//---------------------------------------------------------------------------------------------------------------
//
//  HAUD 2025.02.24
//
//  - EXAMPLE, change, adapt, use
//  -----------------------------
//  - processes and top level workflow examples
//  - based on fb_Instance for processes
//  - fb_Application as top level control for starting, stopping, restarting etc..
//---------------------------------------------------------------------------------------------------------------
PROGRAM MAIN_APP
VAR
  eInit                       : E_PROGRESS;   // application startup state info
  nProcess                    : uint;

  tonWriteLog                 : Tc2_Standard.TON;
  tWriteLog                   : TIME := T#1S;

  stMsg                       : ST_Message;

  _nBufferOutfeedTarget       : ARRAY[1..2] OF E_INSTANCE;
  _nStnFrst                   : UDINT;

  eMsgState                   : e_message_state;
  eMsgProgress                : E_PROGRESS;
END_VAR

//-----------------------------------------------------------------------------------------------------------------
//-----------------------------------------------------------------------------------------------------------------
// check for MAIN.eInit
//  - wait for fb_TransportUnit to be fully started up
//-----------------------------------------------------------------------------------------------------------------
IF NOT (MAIN.eInit = E_PROGRESS.PROGRESS_DONE) 
THEN 
  eInit                                                     := E_PROGRESS.PROGRESS_INVALID; 
  FOR nProcess := E_INSTANCE.BUFFER_INFEED TO MAX_PROCESS
  DO
    GVL_MSG.MessageLevelProcess[nProcess]                   := GVL_MSG.MessageLevel;
  END_FOR
  //ApplicationMain.MessageLevel                              := GVL_MSG.MessageLevel;

  RETURN; 
END_IF
//-----------------------------------------------------------------------------------------------------------------
// set MAIN_APP message device identification
//-----------------------------------------------------------------------------------------------------------------
stMsg.eDevice                                               := e_Device.Application;
//-----------------------------------------------------------------------------------------------------------------
//-----------------------------------------------------------------------------------------------------------------
//-----------------------------------------------------------------------------------------------------------------
// /assign dataflow
//-----------------------------------------------------------------------------------------------------------------
FOR nProcess := 1 TO MAX_PROCESS
DO
  // identification for inter-process-commands and process ST_MESSAGE.eDevice
  GVL_APPLICATION.ProcessCollector[nProcess].ProcessId      :=    nProcess;

  // linked list for you to use for inter-process-commands (start trigger, exit trigger..)
  GVL_APPLICATION.ItfProcessList[nProcess]                  :=    GVL_APPLICATION.ProcessList[nProcess];

  // give reference of all XtsStations to every process; range of process must be set at startup (see action Init())
  GVL_APPLICATION.ProcessCollector[nProcess].StationCtrl    REF=  GVL_XTS.StationCtrl;
  GVL_APPLICATION.ProcessCollector[nProcess].StationState   REF=  GVL_XTS.StationState;

  GVL_APPLICATION.ProcessCollector[nProcess].MoverInfo      REF=  GVL_XTS.MoverInfo;

  // global interfaces for you to use in your process function blocks
  GVL_APPLICATION.ItfProcessCollector[nProcess]             :=    GVL_APPLICATION.ProcessCollector[nProcess];
END_FOR
//-----------------------------------------------------------------------------------------------------------------
//-----------------------------------------------------------------------------------------------------------------
//-----------------------------------------------------------------------------------------------------------------
//  process instances
//-----------------------------------------------------------------------------------------------------------------
GVL_APPLICATION.TicketControl.ItfList                          :=    GVL_APPLICATION.TicketList;
GVL_APPLICATION.TicketControl.Ctrl                             REF=  GVL_APPLICATION.TicketListControl;
GVL_APPLICATION.TicketControl.State                            REF=  GVL_APPLICATION.TicketListState;
GVL_APPLICATION.TicketControl.NodeDataInput                    REF=  GVL_APPLICATION.TicketListDataInput;
GVL_APPLICATION.TicketControl.NodeDataOutput                   REF=  GVL_APPLICATION.TicketListDataOutput;
GVL_APPLICATION.TicketControl.MessageLevel                     :=    GVL_MSG.MessageLevelProcess[e_instance.PROCESS_CONDUCTOR];

GVL_APPLICATION.ProcessConductor.TicketLinkedList           :=    GVL_APPLICATION.TicketList;
GVL_APPLICATION.ProcessConductor.InstanceCtrl               REF=  GVL_APPLICATION.InstanceCtrl;
GVL_APPLICATION.ProcessConductor.InstanceState              REF=  GVL_APPLICATION.InstanceState;
GVL_APPLICATION.ProcessConductor.MessageLevel               :=    GVL_MSG.MessageLevelProcess[e_instance.PROCESS_CONDUCTOR];

GVL_APPLICATION.BufferInfeed.InstanceCtrl                   REF=  GVL_APPLICATION.InstanceCtrl;
GVL_APPLICATION.BufferInfeed.InstanceState                  REF=  GVL_APPLICATION.InstanceState;
GVL_APPLICATION.BufferInfeed.MessageLevel                   :=    GVL_MSG.MessageLevelProcess[e_instance.BUFFER_INFEED];
                                                            
GVL_APPLICATION.Infeed.InstanceCtrl                         REF=  GVL_APPLICATION.InstanceCtrl;
GVL_APPLICATION.Infeed.InstanceState                        REF=  GVL_APPLICATION.InstanceState;
GVL_APPLICATION.Infeed.MessageLevel                         :=    E_MessageType.eMessageSentient; //GVL_MSG.MessageLevelProcess[e_instance.INFEED];
                                                            
GVL_APPLICATION.BufferOutfeed.InstanceCtrl                  REF=  GVL_APPLICATION.InstanceCtrl;
GVL_APPLICATION.BufferOutfeed.InstanceState                 REF=  GVL_APPLICATION.InstanceState;
GVL_APPLICATION.BufferOutfeed.MessageLevel                  :=    GVL_MSG.MessageLevelProcess[e_instance.BUFFER_OUTFEED];
                                                            
GVL_APPLICATION.Outfeed_R1.InstanceCtrl                     REF=  GVL_APPLICATION.InstanceCtrl;
GVL_APPLICATION.Outfeed_R1.InstanceState                    REF=  GVL_APPLICATION.InstanceState;
GVL_APPLICATION.Outfeed_R1.MessageLevel                     :=    GVL_MSG.MessageLevelProcess[e_instance.OUTFEED_ROBOT_R1];
                                                            
GVL_APPLICATION.Outfeed_R2.InstanceCtrl                     REF=  GVL_APPLICATION.InstanceCtrl;
GVL_APPLICATION.Outfeed_R2.InstanceState                    REF=  GVL_APPLICATION.InstanceState;
GVL_APPLICATION.Outfeed_R2.MessageLevel                     :=    GVL_MSG.MessageLevelProcess[e_instance.OUTFEED_ROBOT_R2];
                                                            
GVL_APPLICATION.SenderFast.InstanceCtrl                     REF=  GVL_APPLICATION.InstanceCtrl;
GVL_APPLICATION.SenderFast.InstanceState                    REF=  GVL_APPLICATION.InstanceState;
GVL_APPLICATION.SenderFast.MessageLevel                     :=    GVL_MSG.MessageLevelProcess[e_instance.SENDER_FAST];
                                                            
GVL_APPLICATION.SenderBufferInfeed.InstanceCtrl             REF=  GVL_APPLICATION.InstanceCtrl;
GVL_APPLICATION.SenderBufferInfeed.InstanceState            REF=  GVL_APPLICATION.InstanceState;
GVL_APPLICATION.SenderBufferInfeed.MessageLevel             :=    GVL_MSG.MessageLevelProcess[e_instance.SENDER_BUFFER_INFEED];
//-----------------------------------------------------------------------------------------------------------------
//-----------------------------------------------------------------------------------------------------------------
//-----------------------------------------------------------------------------------------------------------------
//  main application class
//-----------------------------------------------------------------------------------------------------------------
(*
GVL_APPLICATION.ApplicationMain.Ctrl                        REF=  GVL_APPLICATION.AppControl;
GVL_APPLICATION.ApplicationMain.State                       REF=  GVL_APPLICATION.AppState;
GVL_APPLICATION.ApplicationMain.CollectorInterface          REF=  GVL_APPLICATION.ItfProcessCollector;
GVL_APPLICATION.ApplicationMain.ProcessLinkedLists          REF=  GVL_APPLICATION.ItfProcessList;
GVL_APPLICATION.ApplicationMain.XtsTransportCtrl            REF=  GVL_XTS.XtsTransportCtrl;
GVL_APPLICATION.ApplicationMain.XtsTransportState           REF=  GVL_XTS.XtsTransportState;
GVL_APPLICATION.ApplicationMain.InstanceCtrl                REF=  GVL_APPLICATION.InstanceCtrl;
GVL_APPLICATION.ApplicationMain.InstanceState               REF=  GVL_APPLICATION.InstanceState;
*)
//-----------------------------------------------------------------------------------------------------------------
//-----------------------------------------------------------------------------------------------------------------
//-----------------------------------------------------------------------------------------------------------------
// assign dataflow/
//-----------------------------------------------------------------------------------------------------------------
//-----------------------------------------------------------------------------------------------------------------
//-----------------------------------------------------------------------------------------------------------------
//-----------------------------------------------------------------------------------------------------------------
//  /STARTUP
//
// startup procedure for application
//  - connects processes and XtsStations
//-----------------------------------------------------------------------------------------------------------------
CASE eInit
OF
  E_PROGRESS.PROGRESS_INVALID:                // first cycle startup
    //---------------------------------------------------------------------------------------------------------------
    // first cycle startup
    // - wait for extern to give the command, if we are waiting here MAIN is ready, extern can see that
    //---------------------------------------------------------------------------------------------------------------
    GVL_MSG.ApplicationMessageCtrl.Cmd        := E_MESSAGE_CTRL.MSG_CTRL_NULL;
    eInit                                     := E_PROGRESS.PROGRESS_INIT;

  E_PROGRESS.PROGRESS_INIT:
    //---------------------------------------------------------------------------------------------------------------
    // wait for extern to select valid variant
    //---------------------------------------------------------------------------------------------------------------
    CASE GVL_APPLICATION.AppControl.Variant
    OF
      E_APP_VARIANT.VARIANT_OUTPUT_24:
        eInit                                 := E_PROGRESS.PROGRESS_BUSY;
        ProcessInit_R1R2();
  
        stMsg.eType                           := E_MessageType.eMessageInfo;
        stMsg.eSubdevice                      := e_Subdevice.General;
        stMsg.iErrorNumber                    := eInit;
        stMsg.sText                           := concat('MAIN_APP.eInit: ', TO_STRING(eInit));
        stMsg.sText                           := concat(stMsg.sText, ': ');
        stMsg.sText                           := concat(stMsg.sText, TO_STRING(E_INSTANCE.OUTFEED_ROBOT_R1));
        stMsg.sText                           := concat(stMsg.sText, ': ');
        stMsg.sText                           := concat(stMsg.sText, TO_STRING(E_INSTANCE.OUTFEED_ROBOT_R2));
        f_MessageSet(stMsg);

      E_APP_VARIANT.VARIANT_OUTPUT_CLAMP:
        eInit                                 := E_PROGRESS.PROGRESS_BUSY;
        ProcessInit_CLAMP();
  
        stMsg.eType                           := E_MessageType.eMessageInfo;
        stMsg.eSubdevice                      := e_Subdevice.General;
        stMsg.iErrorNumber                    := eInit;
        stMsg.sText                           := concat('MAIN_APP.eInit: ', TO_STRING(eInit));
        stMsg.sText                           := concat(stMsg.sText, ': ');
        stMsg.sText                           := concat(stMsg.sText, TO_STRING(E_INSTANCE.OUTFEED_ROBOT_R1));
        f_MessageSet(stMsg);
    END_CASE

  E_PROGRESS.PROGRESS_BUSY:
    //---------------------------------------------------------------------------------------------------------------
    // first cycle startup of all instances
    //---------------------------------------------------------------------------------------------------------------
    GVL_MSG.ApplicationMessageCtrl.Cmd        := E_MESSAGE_CTRL.MSG_CTRL_INIT;

    IF (GVL_MSG.ApplicationMessageState.State = E_MESSAGE_STATE.MSG_STATE_INIT + E_PROGRESS.PROGRESS_DONE)
    THEN
      eInit                                   := E_PROGRESS.PROGRESS_STARTUP;
    END_IF

  E_PROGRESS.PROGRESS_STARTUP:
    IF GVL_MSG.ApplicationMessageData.FileCreated
    THEN
      eInit                                   := E_PROGRESS.PROGRESS_DONE;
      GVL_MSG.ApplicationMessageCtrl.Cmd      := E_MESSAGE_CTRL.MSG_CTRL_NULL;
    END_IF
END_CASE
GVL_APPLICATION.AppState.AppInit              := eInit;
//-----------------------------------------------------------------------------------------------------------------
//-----------------------------------------------------------------------------------------------------------------
// STARTUP/
//-----------------------------------------------------------------------------------------------------------------
//-----------------------------------------------------------------------------------------------------------------
//-----------------------------------------------------------------------------------------------------------------
// /cyclic calls
//-----------------------------------------------------------------------------------------------------------------
//GVL_APPLICATION.ApplicationMain();

GVL_APPLICATION.TicketControl();

GVL_APPLICATION.ProcessConductor();
GVL_APPLICATION.BufferInfeed();
GVL_APPLICATION.Infeed();
GVL_APPLICATION.BufferOutfeed();
GVL_APPLICATION.Outfeed_R1();
GVL_APPLICATION.Outfeed_R2();
GVL_APPLICATION.SenderFast();
GVL_APPLICATION.SenderBufferInfeed();

FOR nProcess := 1 TO MAX_PROCESS
DO
  // cyclic interface check with XtsStations
  GVL_APPLICATION.ItfProcessCollector[nProcess].Cycle();    // collect XtsStation states, 
                                                            // manage ctrl input from process to XtsStations
END_FOR
//-----------------------------------------------------------------------------------------------------------------
//############################################################################
// /logging
//############################################################################
GVL_MSG.ApplicationMessageData.Ctrl           REF= GVL_MSG.ApplicationMessageCtrl;
GVL_MSG.ApplicationMessageData.State          REF= GVL_MSG.ApplicationMessageState;

GVL_MSG.ApplicationMessageData.MessageIndex   REF= GVL_MSG.MessageApplicationIndex;
GVL_MSG.ApplicationMessageData.ErrorIndex     REF= GVL_MSG.MessageApplicationError;

GVL_MSG.ApplicationMessageData.DirRoot        :=   ADR(GVL_MSG.LOG_DIR);
GVL_MSG.ApplicationMessageData.FileRoot       :=   ADR(GVL_MSG.LOG_FILE_APP);

GVL_MSG.ApplicationMessageData.MsgList        :=   ADR(GVL_MSG.ApplicationMessages);
GVL_MSG.ApplicationMessageData.LocalTime      :=   ADR(GVL_MSG.dtLocalTime);

GVL_MSG.ApplicationMessageData();

eMsgState                                     := f_GetState   (GVL_MSG.ApplicationMessageState.State);
eMsgProgress                                  := f_GetProgress(GVL_MSG.ApplicationMessageState.State);


CASE eMsgState
OF
  E_MESSAGE_STATE.MSG_STATE_NULL:
    CASE eMsgProgress
    OF
      E_PROGRESS.PROGRESS_INVALID:
        IF (GVL_MSG.MessageApplicationIndex > GVL_MSG.MAX_MESSAGE/100) OR
           (GVL_MSG.MessageApplicationError > 0)
        THEN
          GVL_MSG.ApplicationMessageCtrl.Cmd  := E_MESSAGE_CTRL.MSG_CTRL_WRITE;
        END_IF
    END_CASE

  E_MESSAGE_STATE.MSG_STATE_WRITE:
    CASE eMsgProgress
    OF
      E_PROGRESS.PROGRESS_ERROR,
      E_PROGRESS.PROGRESS_DONE:
        GVL_MSG.ApplicationMessageCtrl.Cmd    := E_MESSAGE_CTRL.MSG_CTRL_NULL;
    END_CASE

ELSE
    CASE eMsgProgress
    OF
      E_PROGRESS.PROGRESS_DONE:
        GVL_MSG.ApplicationMessageCtrl.Cmd    := E_MESSAGE_CTRL.MSG_CTRL_NULL;
    END_CASE
END_CASE
//############################################################################
// logging/
//############################################################################

ACTION ProcessInit_CLAMP:
//*************************************************************************************************************
//
// build configuration for Instances and ProcessInterfaces
//
//*************************************************************************************************************
//*************************************************************************************************************
// - ProcessConductor : Instance with connection to a cyclic linked list 
//                      Here does The Ticket with target processId and bitmask arrive 
//                      this instance forwards the ticket to its destination
//                        destination is BufferInfeed
//-------------------------------------------------------------------------------------------------------------
// whoami
//
// ticket box - transfersystem drops ticket
//-------------------------------------------------------------------------------------------------------------
ProcessConductor.ProcessId                := ProcessCollector[E_INSTANCE.PROCESS_CONDUCTOR].ProcessId;
ProcessConductor.CollectorInterface       := ItfProcessCollector;
ProcessConductor.ProcessLinkedLists       := ItfProcessList;

//*************************************************************************************************************
// - BufferInfeed     : single XtsStation which looks for input trigger from transfersystem, 
//                      transfersystem writes positions of XtsStations to be used at Infeed. 
//                      BufferInfeed is writing ItfProcessCollector[BufferInfeed.ProcessTarget].ActivateStation 
//                        for BufferInfeed target (Infeed / 12 XtsStations).
//                      BufferInfeed sends required amount of movers to WaitPos of XtsStations 
//                        of BufferInfeed target (Infeed / 12 XtsStations).
//-------------------------------------------------------------------------------------------------------------
// whoami
//
// process target (Infeed / 12 XtsStations)
//-------------------------------------------------------------------------------------------------------------
BufferInfeed.ProcessId                    := ProcessCollector[E_INSTANCE.BUFFER_INFEED].ProcessId;
BufferInfeed.ProcessTarget                := ProcessCollector[E_INSTANCE.INFEED].ProcessId;
BufferInfeed.CollectorInterface           := ItfProcessCollector;
BufferInfeed.ProcessLinkedLists           := ItfProcessList;
//-------------------------------------------------------------------------------------------------------------
// configure range of XtsStations for process
//
// see MAIN.StationParameterInit() for positions and dyn constraints
//-------------------------------------------------------------------------------------------------------------
ItfProcessCollector[BufferInfeed.ProcessId].StationFirst  := 53;
ItfProcessCollector[BufferInfeed.ProcessId].StationLast   := 53;

_nStnFrst                                 := ProcessCollector[BufferInfeed.ProcessId].StationFirst;
BufferInfeed.CheckPosition                := 15.0;

//-------------------------------------------------------------------------------------------------------------
//-------------------------------------------------------------------------------------------------------------
//*************************************************************************************************************
//*************************************************************************************************************
// - Infeed         : 12 XtsStations for transfersystem to unload
//                    Infeed is pulling in the movers according to list entry from BufferInfeed
//                    one stop only
//                    must be checked for all mover standstill in PosStop[1] of each XtsStation
//                    must be released by handshake from transfersystem (this is done by a TON for now)
//-------------------------------------------------------------------------------------------------------------
// whoami
//
// process target (BufferOutfeed / 1 XtsStation)
// TODO: 
//    configure infeed target for OUTFEED_CLAMP (12 XtsStations)
//    Infeed.ProcessTarget  := ProcessCollector[E_INSTANCE.OUTFEED_CLAMP].ProcessId;
//-------------------------------------------------------------------------------------------------------------
Infeed.ProcessId                          := ProcessCollector[E_INSTANCE.INFEED].ProcessId;
Infeed.ProcessTarget                      := ProcessCollector[E_INSTANCE.BUFFER_OUTFEED].ProcessId;
Infeed.CollectorInterface                 := ItfProcessCollector;
Infeed.ProcessLinkedLists                 := ItfProcessList;
//-------------------------------------------------------------------------------------------------------------
// configure range of XtsStations for process
//
// see MAIN.StationParameterInit() for positions and dyn constraints
//-------------------------------------------------------------------------------------------------------------
ItfProcessCollector[Infeed.ProcessId].StationFirst        :=  1;
ItfProcessCollector[Infeed.ProcessId].StationLast         := 12;
//-------------------------------------------------------------------------------------------------------------
//-------------------------------------------------------------------------------------------------------------
//*************************************************************************************************************
//*************************************************************************************************************
// - BufferOutfeed  : single XtsStation which distributes movers to specified range 
//                    Infeed sends all movers here 
//                    BufferOutfeed ensures that OutputR2 and OutputR1 have 12 movers each for every job
//                    BufferOutfeed checks if the Queue of this single XtsStation is empty or not
//-------------------------------------------------------------------------------------------------------------
// whoami
//
// process target (Outfeed (OutfeedR2 & OutfeedR1) / 24 XtsStations)
//
//  - optional process target (Outfeed 12 XtsStations)
//-------------------------------------------------------------------------------------------------------------
_nBufferOutfeedTarget[1] := E_INSTANCE.OUTFEED_ROBOT_R1;
_nBufferOutfeedTarget[2] := E_INSTANCE.OUTFEED_ROBOT_R1;

BufferOutfeed.ProcessId              := E_INSTANCE.BUFFER_OUTFEED;
BufferOutfeed.ProcessTarget          := _nBufferOutfeedTarget; 
BufferOutfeed.CollectorInterface     := ItfProcessCollector;
BufferOutfeed.ProcessLinkedLists     := ItfProcessList;
//-------------------------------------------------------------------------------------------------------------
// configure range of XtsStations for process
//
// see MAIN.StationParameterInit() for positions and dyn constraints
//-------------------------------------------------------------------------------------------------------------
ItfProcessCollector[BufferOutfeed.ProcessId].StationFirst  := 25;
ItfProcessCollector[BufferOutfeed.ProcessId].StationLast   := 25;

_nStnFrst                                 := ProcessCollector[BufferOutfeed.ProcessId].StationFirst;
BufferOutfeed.CheckPosition          := 2250.0;
//-------------------------------------------------------------------------------------------------------------
//-------------------------------------------------------------------------------------------------------------
//*************************************************************************************************************
//*************************************************************************************************************
// - Outfeed_R1  : 12 XtsStations for Robot 
//                    All XtsStations must be filled before robot can start 
//                    affter process all movers are sent to Sender process (high speed for the way back)
//                     
//                    
//-------------------------------------------------------------------------------------------------------------
// whoami
//
// process target (SenderFast / 1 XtsStation)
//-------------------------------------------------------------------------------------------------------------
Outfeed_R1.ProcessId                      := E_INSTANCE.OUTFEED_ROBOT_R1;
Outfeed_R1.ProcessTarget                  := ProcessCollector[E_INSTANCE.SENDER_FAST].ProcessId;
Outfeed_R1.CollectorInterface             := ItfProcessCollector;
Outfeed_R1.ProcessLinkedLists             := ItfProcessList;
//-------------------------------------------------------------------------------------------------------------
// configure range of XtsStations for process
//
// see MAIN.StationParameterInit() for positions and dyn constraints
//-------------------------------------------------------------------------------------------------------------
ItfProcessCollector[Outfeed_R1.ProcessId].StationFirst  := 13;
ItfProcessCollector[Outfeed_R1.ProcessId].StationLast   := 24;

_nStnFrst                                 := ProcessCollector[Outfeed_R1.ProcessId].StationFirst;
Outfeed_R1.CheckPosition                  := 2750.0;
//-------------------------------------------------------------------------------------------------------------
//-------------------------------------------------------------------------------------------------------------
//*************************************************************************************************************
//*************************************************************************************************************
// - Outfeed_R2  : 12 XtsStations for Robot 
//                    All XtsStations must be filled before robot can start 
//                    affter process all movers are sent to Sender process (high speed for the way back)
//                     
//                    
//-------------------------------------------------------------------------------------------------------------
// whoami
//
// process target (SenderFast / 1 XtsStation)
//-------------------------------------------------------------------------------------------------------------
Outfeed_R2.ProcessId                      := E_INSTANCE.OUTFEED_ROBOT_R2;
Outfeed_R2.ProcessTarget                  := ProcessCollector[E_INSTANCE.SENDER_FAST].ProcessId;
Outfeed_R2.CollectorInterface             := ItfProcessCollector;
Outfeed_R2.ProcessLinkedLists             := ItfProcessList;
//-------------------------------------------------------------------------------------------------------------
// configure range of XtsStations for process
//
// see MAIN.StationParameterInit() for positions and dyn constraints
//-------------------------------------------------------------------------------------------------------------
ItfProcessCollector[Outfeed_R2.ProcessId].StationFirst  := 38;
ItfProcessCollector[Outfeed_R2.ProcessId].StationLast   := 49;

_nStnFrst                                 := ProcessCollector[Outfeed_R2.ProcessId].StationFirst;
Outfeed_R2.CheckPosition                  := 6000.0;
//-------------------------------------------------------------------------------------------------------------
//-------------------------------------------------------------------------------------------------------------
//*************************************************************************************************************
//*************************************************************************************************************
// - SenderFast  : 1 XtsStation 
//                    movers are handled when entering position area 
//                    movers are accelerated to max speed
//                    movers do not stop here
//                    
//-------------------------------------------------------------------------------------------------------------
// whoami
//
// process target (SenderBufferInfeed / 1 XtsStation)
//-------------------------------------------------------------------------------------------------------------
SenderFast.ProcessId                      := E_INSTANCE.SENDER_FAST;
SenderFast.ProcessTarget                  := ProcessCollector[E_INSTANCE.SENDER_BUFFER_INFEED].ProcessId;
SenderFast.CollectorInterface             := ItfProcessCollector;
SenderFast.ProcessLinkedLists             := ItfProcessList;
//-------------------------------------------------------------------------------------------------------------
// configure range of XtsStations for process
//
// see MAIN.StationParameterInit() for positions and dyn constraints
//-------------------------------------------------------------------------------------------------------------
ItfProcessCollector[SenderFast.ProcessId].StationFirst  := 51;
ItfProcessCollector[SenderFast.ProcessId].StationLast   := 51;

_nStnFrst                                 := ProcessCollector[SenderFast.ProcessId].StationFirst;
SenderFast.CheckPosition                  := GVL_XTS.StationParameter[_nStnFrst].rPosWait - 500.0;
//-------------------------------------------------------------------------------------------------------------
//-------------------------------------------------------------------------------------------------------------
//*************************************************************************************************************
//*************************************************************************************************************
// - SenderBufferInfeed  : 1 XtsStation 
//                    movers are handled when entering position area 
//                    movers are sent to BufferInfeed, so that BufferInfeed has 12 mover ready
//                    movers do stop here, wait until there is room for movers
//                    
//-------------------------------------------------------------------------------------------------------------
// whoami
//
// process target (SenderBufferInfeed / 1 XtsStation)
//-------------------------------------------------------------------------------------------------------------
SenderBufferInfeed.ProcessId              := E_INSTANCE.SENDER_BUFFER_INFEED;
SenderBufferInfeed.ProcessTarget          := ProcessCollector[E_INSTANCE.BUFFER_INFEED].ProcessId;
SenderBufferInfeed.CollectorInterface     := ItfProcessCollector;
SenderBufferInfeed.ProcessLinkedLists     := ItfProcessList;
//-------------------------------------------------------------------------------------------------------------
// configure range of XtsStations for process
//
// see MAIN.StationParameterInit() for positions and dyn constraints
//-------------------------------------------------------------------------------------------------------------
ItfProcessCollector[SenderBufferInfeed.ProcessId].StationFirst  := 52;
ItfProcessCollector[SenderBufferInfeed.ProcessId].StationLast   := 52;

_nStnFrst                                 := ProcessCollector[SenderBufferInfeed.ProcessId].StationFirst;
SenderBufferInfeed.CheckPosition          := GVL_XTS.StationParameter[_nStnFrst].rPosWait - 250.0;
//-------------------------------------------------------------------------------------------------------------
//-------------------------------------------------------------------------------------------------------------
//*************************************************************************************************************
END_ACTION

ACTION ProcessInit_R1R2:
//*************************************************************************************************************
//
// build configuration for Instances and ProcessInterfaces
//
//*************************************************************************************************************
//*************************************************************************************************************
// - ProcessConductor : Instance with connection to a cyclic linked list 
//                      Here does The Ticket with target processId and bitmask arrive 
//                      this instance forwards the ticket to its destination
//                        destination is BufferInfeed
//-------------------------------------------------------------------------------------------------------------
// whoami
//
// ticket box - transfersystem drops ticket
//-------------------------------------------------------------------------------------------------------------
ProcessConductor.ProcessId                := ProcessCollector[E_INSTANCE.PROCESS_CONDUCTOR].ProcessId;
ProcessConductor.CollectorInterface       := ItfProcessCollector;
ProcessConductor.ProcessLinkedLists       := ItfProcessList;

//*************************************************************************************************************
// - BufferInfeed     : single XtsStation which looks for input trigger from transfersystem, 
//                      transfersystem writes positions of XtsStations to be used at Infeed. 
//                      BufferInfeed is writing ItfProcessCollector[BufferInfeed.ProcessTarget].ActivateStation 
//                        for BufferInfeed target (Infeed / 12 XtsStations).
//                      BufferInfeed sends required amount of movers to WaitPos of XtsStations 
//                        of BufferInfeed target (Infeed / 12 XtsStations).
//-------------------------------------------------------------------------------------------------------------
// whoami
//
// process target (Infeed / 12 XtsStations)
//-------------------------------------------------------------------------------------------------------------
BufferInfeed.ProcessId                    := ProcessCollector[E_INSTANCE.BUFFER_INFEED].ProcessId;
BufferInfeed.ProcessTarget                := ProcessCollector[E_INSTANCE.INFEED].ProcessId;
BufferInfeed.CollectorInterface           := ItfProcessCollector;
BufferInfeed.ProcessLinkedLists           := ItfProcessList;
//-------------------------------------------------------------------------------------------------------------
// configure range of XtsStations for process
//
// see MAIN.StationParameterInit() for positions and dyn constraints
//-------------------------------------------------------------------------------------------------------------
ItfProcessCollector[BufferInfeed.ProcessId].StationFirst  := 53;
ItfProcessCollector[BufferInfeed.ProcessId].StationLast   := 53;

_nStnFrst                                 := ProcessCollector[BufferInfeed.ProcessId].StationFirst;
BufferInfeed.CheckPosition                := 15.0;

//-------------------------------------------------------------------------------------------------------------
//-------------------------------------------------------------------------------------------------------------
//*************************************************************************************************************
//*************************************************************************************************************
// - Infeed         : 12 XtsStations for transfersystem to unload
//                    Infeed is pulling in the movers according to list entry from BufferInfeed
//                    one stop only
//                    must be checked for all mover standstill in PosStop[1] of each XtsStation
//                    must be released by handshake from transfersystem (this is done by a TON for now)
//-------------------------------------------------------------------------------------------------------------
// whoami
//
// process target (BufferOutfeed / 1 XtsStation)
// TODO: 
//    configure infeed target for OUTFEED_CLAMP (12 XtsStations)
//    Infeed.ProcessTarget  := ProcessCollector[E_INSTANCE.OUTFEED_CLAMP].ProcessId;
//-------------------------------------------------------------------------------------------------------------
Infeed.ProcessId                          := ProcessCollector[E_INSTANCE.INFEED].ProcessId;
Infeed.ProcessTarget                      := ProcessCollector[E_INSTANCE.BUFFER_OUTFEED].ProcessId;
Infeed.CollectorInterface                 := ItfProcessCollector;
Infeed.ProcessLinkedLists                 := ItfProcessList;
//-------------------------------------------------------------------------------------------------------------
// configure range of XtsStations for process
//
// see MAIN.StationParameterInit() for positions and dyn constraints
//-------------------------------------------------------------------------------------------------------------
ItfProcessCollector[Infeed.ProcessId].StationFirst        :=  1;
ItfProcessCollector[Infeed.ProcessId].StationLast         := 12;
//-------------------------------------------------------------------------------------------------------------
//-------------------------------------------------------------------------------------------------------------
//*************************************************************************************************************
//*************************************************************************************************************
// - BufferOutfeed  : single XtsStation which distributes movers to specified range 
//                    Infeed sends all movers here 
//                    BufferOutfeed ensures that OutputR2 and OutputR1 have 12 movers each for every job
//                    BufferOutfeed checks if the Queue of this single XtsStation is empty or not
//-------------------------------------------------------------------------------------------------------------
// whoami
//
// process target (Outfeed (OutfeedR2 & OutfeedR1) / 24 XtsStations)
//
//  - optional process target (Outfeed 12 XtsStations)
//-------------------------------------------------------------------------------------------------------------
_nBufferOutfeedTarget[1] := E_INSTANCE.OUTFEED_ROBOT_R1;
_nBufferOutfeedTarget[2] := E_INSTANCE.OUTFEED_ROBOT_R2;

BufferOutfeed.ProcessId              := E_INSTANCE.BUFFER_OUTFEED;
BufferOutfeed.ProcessTarget          := _nBufferOutfeedTarget; 
BufferOutfeed.CollectorInterface     := ItfProcessCollector;
BufferOutfeed.ProcessLinkedLists     := ItfProcessList;
//-------------------------------------------------------------------------------------------------------------
// configure range of XtsStations for process
//
// see MAIN.StationParameterInit() for positions and dyn constraints
//-------------------------------------------------------------------------------------------------------------
ItfProcessCollector[BufferOutfeed.ProcessId].StationFirst  := 25;
ItfProcessCollector[BufferOutfeed.ProcessId].StationLast   := 25;

_nStnFrst                                 := ProcessCollector[BufferOutfeed.ProcessId].StationFirst;
BufferOutfeed.CheckPosition          := 2500.0;
//-------------------------------------------------------------------------------------------------------------
//-------------------------------------------------------------------------------------------------------------
//*************************************************************************************************************
//*************************************************************************************************************
// - Outfeed_R1  : 12 XtsStations for Robot 
//                    All XtsStations must be filled before robot can start 
//                    affter process all movers are sent to Sender process (high speed for the way back)
//                     
//                    
//-------------------------------------------------------------------------------------------------------------
// whoami
//
// process target (SenderFast / 1 XtsStation)
//-------------------------------------------------------------------------------------------------------------
Outfeed_R1.ProcessId                      := E_INSTANCE.OUTFEED_ROBOT_R1;
Outfeed_R1.ProcessTarget                  := ProcessCollector[E_INSTANCE.SENDER_FAST].ProcessId;
Outfeed_R1.CollectorInterface             := ItfProcessCollector;
Outfeed_R1.ProcessLinkedLists             := ItfProcessList;
//-------------------------------------------------------------------------------------------------------------
// configure range of XtsStations for process
//
// see MAIN.StationParameterInit() for positions and dyn constraints
//-------------------------------------------------------------------------------------------------------------
ItfProcessCollector[Outfeed_R1.ProcessId].StationFirst  := 26;
ItfProcessCollector[Outfeed_R1.ProcessId].StationLast   := 37;

_nStnFrst                                 := ProcessCollector[Outfeed_R1.ProcessId].StationFirst;
Outfeed_R1.CheckPosition                  := 6000.0;
//-------------------------------------------------------------------------------------------------------------
//-------------------------------------------------------------------------------------------------------------
//*************************************************************************************************************
//*************************************************************************************************************
// - Outfeed_R2  : 12 XtsStations for Robot 
//                    All XtsStations must be filled before robot can start 
//                    affter process all movers are sent to Sender process (high speed for the way back)
//                     
//                    
//-------------------------------------------------------------------------------------------------------------
// whoami
//
// process target (SenderFast / 1 XtsStation)
//-------------------------------------------------------------------------------------------------------------
Outfeed_R2.ProcessId                      := E_INSTANCE.OUTFEED_ROBOT_R2;
Outfeed_R2.ProcessTarget                  := ProcessCollector[E_INSTANCE.SENDER_FAST].ProcessId;
Outfeed_R2.CollectorInterface             := ItfProcessCollector;
Outfeed_R2.ProcessLinkedLists             := ItfProcessList;
//-------------------------------------------------------------------------------------------------------------
// configure range of XtsStations for process
//
// see MAIN.StationParameterInit() for positions and dyn constraints
//-------------------------------------------------------------------------------------------------------------
ItfProcessCollector[Outfeed_R2.ProcessId].StationFirst  := 38;
ItfProcessCollector[Outfeed_R2.ProcessId].StationLast   := 49;

_nStnFrst                                 := ProcessCollector[Outfeed_R2.ProcessId].StationFirst;
Outfeed_R2.CheckPosition                  := 6000.0;
//-------------------------------------------------------------------------------------------------------------
//-------------------------------------------------------------------------------------------------------------
//*************************************************************************************************************
//*************************************************************************************************************
// - SenderFast  : 1 XtsStation 
//                    movers are handled when entering position area 
//                    movers are accelerated to max speed
//                    movers do not stop here
//                    
//-------------------------------------------------------------------------------------------------------------
// whoami
//
// process target (SenderBufferInfeed / 1 XtsStation)
//-------------------------------------------------------------------------------------------------------------
SenderFast.ProcessId                      := E_INSTANCE.SENDER_FAST;
SenderFast.ProcessTarget                  := ProcessCollector[E_INSTANCE.SENDER_BUFFER_INFEED].ProcessId;
SenderFast.CollectorInterface             := ItfProcessCollector;
SenderFast.ProcessLinkedLists             := ItfProcessList;
//-------------------------------------------------------------------------------------------------------------
// configure range of XtsStations for process
//
// see MAIN.StationParameterInit() for positions and dyn constraints
//-------------------------------------------------------------------------------------------------------------
ItfProcessCollector[SenderFast.ProcessId].StationFirst  := 51;
ItfProcessCollector[SenderFast.ProcessId].StationLast   := 51;

_nStnFrst                                 := ProcessCollector[SenderFast.ProcessId].StationFirst;
SenderFast.CheckPosition                  := GVL_XTS.StationParameter[_nStnFrst].rPosWait - 500.0;
//-------------------------------------------------------------------------------------------------------------
//-------------------------------------------------------------------------------------------------------------
//*************************************************************************************************************
//*************************************************************************************************************
// - SenderBufferInfeed  : 1 XtsStation 
//                    movers are handled when entering position area 
//                    movers are sent to BufferInfeed, so that BufferInfeed has 12 mover ready
//                    movers do stop here, wait until there is room for movers
//                    
//-------------------------------------------------------------------------------------------------------------
// whoami
//
// process target (SenderBufferInfeed / 1 XtsStation)
//-------------------------------------------------------------------------------------------------------------
SenderBufferInfeed.ProcessId              := E_INSTANCE.SENDER_BUFFER_INFEED;
SenderBufferInfeed.ProcessTarget          := ProcessCollector[E_INSTANCE.BUFFER_INFEED].ProcessId;
SenderBufferInfeed.CollectorInterface     := ItfProcessCollector;
SenderBufferInfeed.ProcessLinkedLists     := ItfProcessList;
//-------------------------------------------------------------------------------------------------------------
// configure range of XtsStations for process
//
// see MAIN.StationParameterInit() for positions and dyn constraints
//-------------------------------------------------------------------------------------------------------------
ItfProcessCollector[SenderBufferInfeed.ProcessId].StationFirst  := 52;
ItfProcessCollector[SenderBufferInfeed.ProcessId].StationLast   := 52;

_nStnFrst                                 := ProcessCollector[SenderBufferInfeed.ProcessId].StationFirst;
SenderBufferInfeed.CheckPosition          := GVL_XTS.StationParameter[_nStnFrst].rPosWait - 1250.0;
//-------------------------------------------------------------------------------------------------------------
//-------------------------------------------------------------------------------------------------------------
//*************************************************************************************************************
END_ACTION

END_PROGRAM

(* stored: Version 1.1.0.1, ProductVersion 3.1.4026.13
   POU MAIN_APP: Id {1c97d90f-7a21-4183-a188-63046e9cbf94}, SpecialFunc None
   Action ProcessInit_CLAMP: Id {4a34d2c2-2306-48d6-9a70-3233cf83d9f2}
   Action ProcessInit_R1R2: Id {1fb39183-07c5-42fa-837d-3255551b6608} *)
